# EPICS substitutions: hugo/source/db/Beckhoff_9XXX/ecmcEL9410.substitutions
file "ecmcEL9410-chX.template"
{
  pattern {CH_ID}
          {01   }
}
